PROGRAM Datos_Variadores
VAR
	Variador_6 :SDO_READ;
	ReadStart :BOOL;
	ReadError :DWORD;
	ReadData :ARRAY[0..255] OF BYTE;
	AuxRPM:u_RPM;
	RPM_6 :INT;
END_VAR



Variador_6(

    StartReading := ReadStart,
    CO_Index := 16#2042,
    CO_SubIndex := 16#5,
    DataLength := 2,
    PortNr := 16#1005,
    ADSNetID:='169.254.25.50.3.1'
    );

IF Variador_6.ReadDataAvailable THEN
    ReadStart := FALSE;
    ReadError := Variador_6.Error;
    ReadData := Variador_6.ReadData;
END_IF
AuxRPM.rpm[0]:=ReadData[0];
AuxRPM.rpm[1]:=ReadData[1];
RPM_6 :=AuxRPM.iRpm;

END_PROGRAM

(* stored: Version 1.1.0.1, ProductVersion 3.1.4024.12
   POU Datos_Variadores: Id {d53b7410-187b-4f15-b0b8-c1963b9f240e}, SpecialFunc None *)
